TYPE ST_ReactivePower :
STRUCT
	ReactivePower_Total		:DINT;
	ReactivePower_L1		:DINT;
	ReactivePower_L2		:DINT;
	ReactivePower_L3		:DINT;
END_STRUCT
END_TYPE

(* stored: Version 1.1.0.1, ProductVersion 3.1.4022.3
   DUT ST_ReactivePower: Id {5c43479f-b4e5-474e-8097-9967817e30ed} *)
